Yaskawa INFORM job: B-3-08279-80-SUB-L.JBI

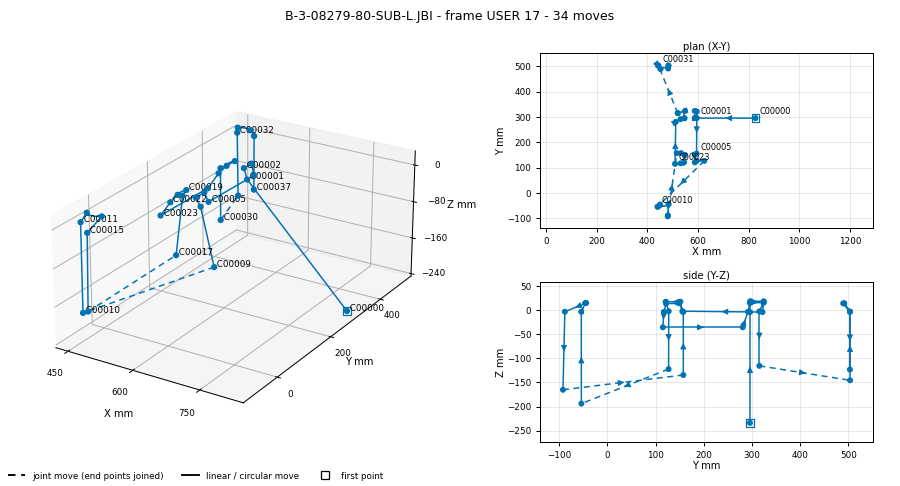
[picture p0: tool path of B-3-08279-80-SUB-L.JBI in frame USER 17, 34 of 38 moves have a stored position in this frame; points joined in program order, loops and branches not executed]
/JOB
//NAME B-3-08279-80-SUB-L
///FOLDERNAME PART_420-08279-80
//POS
///NPOS 38,0,38,0,0,0
///USER 17
///TOOL 4
///POSTYPE USER
///RECTAN
///RCONF 1,0,0,0,0,0,0,0,0,0,0,0,0,0,0,0,0,0,0,0,0,0,0,0
C00000=826.493,295.690,-233.792,-27.8958,11.3049,78.2347
C00001=594.519,295.721,-3.979,-46.5250,6.9320,75.2540
C00002=586.715,296.087,18.419,-46.5244,6.9323,75.2546
C00003=586.699,324.081,18.424,-46.5242,6.9325,75.2557
C00004=594.755,321.720,-3.979,-46.5250,6.9320,75.2540
C00005=593.773,155.478,-2.185,-42.9430,-21.0870,89.6170
C00006=586.962,151.268,17.533,-42.9383,-21.0893,89.6174
C00007=586.958,120.949,17.499,-42.9372,-21.0891,89.6171
C00008=593.773,127.194,-2.185,-42.9430,-21.0870,89.6170
C00009=624.287,126.871,-122.266,-42.9430,-21.0870,89.6170
C00010=439.602,-53.998,-193.900,-6.5584,-44.9787,-116.9694
C00011=440.802,-54.182,-3.282,-6.5590,-44.9790,-116.9690
C00012=449.618,-45.388,15.082,-6.5573,-44.9806,-116.9699
C00013=464.573,-51.760,15.080,-6.5575,-44.9789,-90.5140
C00014=483.194,-44.207,14.751,-6.5596,-44.9771,-55.2507
C00015=480.565,-88.232,-3.329,-6.5583,-44.9788,-55.2558
C00016=479.931,-92.164,-165.151,-6.5577,-44.9788,-55.2551
C00017=515.569,157.432,-134.492,-16.3485,-44.1216,152.7886
C00018=532.609,157.384,-3.682,-16.3490,-44.1220,152.7880
C00019=547.093,148.694,14.622,-12.3664,-44.9876,162.0022
C00020=542.303,136.291,13.860,-16.8317,-44.9292,-164.4086
C00021=544.832,121.690,13.631,-16.5140,-44.7703,-145.3126
C00022=530.621,117.175,-3.669,-16.5140,-44.7720,-151.5720
C00023=508.748,115.031,-35.500,-16.5140,-44.7720,-151.5720
C00024=511.771,280.690,-35.500,3.4420,-44.9790,-154.0720
C00025=530.020,291.566,-3.353,3.4420,-44.9790,-154.0720
C00026=546.591,295.454,15.049,3.6602,-45.0537,-167.8784
C00027=543.113,311.140,15.551,7.8965,-43.2324,176.8605
C00028=547.905,324.077,15.653,15.6707,-44.9801,144.2143
C00029=519.589,315.156,-2.528,16.5470,-44.9790,144.2150
C00030=519.589,315.156,-115.500,16.5470,-44.9790,144.2150
C00031=443.469,503.235,-145.503,28.9250,-36.2220,77.7093
C00032=441.430,503.175,-3.498,16.2188,-41.7424,92.6652
C00033=451.601,489.089,14.088,16.2184,-41.7431,92.6641
C00034=467.002,495.184,14.131,15.7370,-42.8117,71.8233
C00035=481.720,491.356,13.958,13.1213,-43.5296,40.3770
C00036=482.884,503.018,-2.647,12.3290,-43.7170,41.5290
C00037=482.649,502.996,-123.098,12.0361,-43.7836,41.9512
///TOOL 0
///POSTYPE ANGLE
///ANGLE
EC00000=-45.0000
///TOOL 4
EC00001=-45.0000
///TOOL 0
EC00002=-45.0000
EC00003=-45.0000
///TOOL 4
EC00004=-45.0000
EC00005=-45.0000
///TOOL 0
EC00006=-45.0005
EC00007=-45.0005
///TOOL 4
EC00008=-45.0000
EC00009=-45.0000
///TOOL 0
EC00010=-90.0000
///TOOL 4
EC00011=-90.0000
///TOOL 0
EC00012=-90.0000
EC00013=-90.0000
EC00014=-90.0000
EC00015=-90.0000
EC00016=-90.0000
EC00017=-90.0000
///TOOL 4
EC00018=-90.0000
///TOOL 0
EC00019=-90.0000
EC00020=-90.0000
EC00021=-90.0000
///TOOL 4
EC00022=-90.0000
EC00023=-90.0000
EC00024=-90.0000
EC00025=-90.0000
///TOOL 0
EC00026=-90.0000
EC00027=-90.0000
EC00028=-90.0000
///TOOL 4
EC00029=-90.0000
EC00030=-90.0000
///TOOL 0
EC00031=-90.0000
EC00032=-90.0000
EC00033=-90.0000
EC00034=-90.0000
EC00035=-90.0000
///TOOL 4
EC00036=-90.0000
///TOOL 0
EC00037=-90.0000
//INST
///DATE 2021/10/29 11:36
///ATTR SC,RW,RJ
////FRAME USER 17
///GROUP1 RB1
///GROUP2 ST3
NOP
'Path Start: PP9
'Warning, the first motion progra
'mmed for this routine was not a
'joint motion
'The following movement has been
'added. Please update your OCTOPU
'Z simulation.
MOVJ C00000 VJ=100.00  +MOVJ EC00000
SMOVL C00001 V=1250.0  +MOVJ EC00001
SMOVL C00002 V=300.0  +MOVJ EC00002
ARCON ASF#(951)
SMOVL C00003 V=8.5  +MOVJ EC00003
ARCOF AEF#(951)
SMOVL C00004 V=1250.0  +MOVJ EC00004
'Path End
'Path Start: PP15
SMOVL C00005 V=1250.0  +MOVJ EC00005
SMOVL C00006 V=300.0  +MOVJ EC00006
ARCON ASF#(951)
SMOVL C00007  +MOVJ EC00007
ARCOF AEF#(951)
SMOVL C00008 V=1250.0  +MOVJ EC00008
SMOVL C00009 V=1250.0  +MOVJ EC00009
'Path End
'Path Start: PP16
MOVJ C00010 VJ=25.00  +MOVJ EC00010
SMOVL C00011 V=1250.0  +MOVJ EC00011
SMOVC C00012 V=300.0  +MOVJ EC00012
ARCON ASF#(951)
SMOVC C00013 V=8.5  +MOVJ EC00013
SMOVC C00014 V=8.5  +MOVJ EC00014
ARCOF AEF#(951)
SMOVL C00015 V=1250.0  +MOVJ EC00015
SMOVL C00016 V=1250.0  +MOVJ EC00016
'Path End
'Path Start: PP19
MOVJ C00017 VJ=100.00  +MOVJ EC00017
SMOVL C00018 V=1250.0  +MOVJ EC00018
SMOVC C00019 V=300.0  +MOVJ EC00019
ARCON ASF#(951)
SMOVC C00020 V=8.5  +MOVJ EC00020
SMOVC C00021 V=8.5  +MOVJ EC00021
ARCOF AEF#(951)
SMOVL C00022 V=1250.0  +MOVJ EC00022
SMOVL C00023 V=1250.0  +MOVJ EC00023
'Path End
'Path Start: PP20
SMOVL C00024 V=1250.0  +MOVJ EC00024
SMOVL C00025 V=1250.0  +MOVJ EC00025
SMOVC C00026 V=300.0  +MOVJ EC00026
ARCON ASF#(951)
SMOVC C00027 V=8.5  +MOVJ EC00027
SMOVC C00028 V=8.5  +MOVJ EC00028
ARCOF AEF#(951)
SMOVL C00029 V=1250.0  +MOVJ EC00029
SMOVL C00030 V=1250.0  +MOVJ EC00030
'Path End
'Path Start: PP22
MOVJ C00031 VJ=100.00  +MOVJ EC00031
SMOVL C00032 V=1250.0  +MOVJ EC00032
SMOVC C00033 V=300.0  +MOVJ EC00033
ARCON ASF#(951)
SMOVC C00034 V=8.5  +MOVJ EC00034
SMOVC C00035 V=8.5  +MOVJ EC00035
ARCOF AEF#(951)
SMOVL C00036 V=1250.0  +MOVJ EC00036
SMOVL C00037 V=1250.0  +MOVJ EC00037
'Path End
END
